//latching (self-holding) relay circuit
PROGRAM p02_clock
VAR
	M0: BOOL;
END_VAR

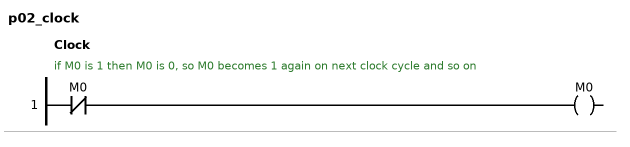
// NETWORK 1: Clock
// if M0 is 1 then M0 is 0, so M0 becomes 1 again on next clock cycle and so on
M0 := NOT M0;

END_PROGRAM

(* stored: Version 1.1.0.1, ProductVersion 3.1.4024.13
   POU p02_clock: Id {50fedffc-eb7f-4705-90e0-7907d160e0f5}, SpecialFunc None *)
